PROGRAM CartControl
VAR
	// cart instance
	m_masterCart :FB_MasterCart;
	
	//cart related UI
	m_cartUIData : ST_CartUIData;
	
	// Output cart status
	m_cartStatus AT%Q* : ST_CartStatus;
	
	// Cart  joint data
	m_cartJointData AT %Q* :ST_CartJointData;
	
	// wait time before cart init for ethercat to be statble 
	m_cartInitWaitTime : LREAL:=0;
	
	// cart init flag
	m_cartInit :BOOL :=FALSE;
	
	m_workHeartTon0 : TON;
	m_workHeartTon1 : TON;
	
END_VAR

// wait communication to be stable
IF(m_cartInitWaitTime<g_robotInitWaitTime) THEN
	m_cartInitWaitTime := m_cartInitWaitTime+g_armCtrlCycleTime;
	RETURN;
END_IF

// cart init
IF m_cartInit =FALSE THEN
	m_masterCart.Init();
	m_cartInit:=TRUE;
END_IF

// input from UI
UIInputProcess();

// cart run
m_masterCart.run(m_cartUIData);

// status/joint data output
m_masterCart.getStatus(m_cartStatus, m_cartJointData);

// tranform data from UI(global variable write by ADS) to ST_UIData
METHOD UIInputProcess : BOOL
VAR_INPUT
END_VAR
//init cart joint postion
IF (GVL_interactUI.Upper_PC_Initial_Finished=FALSE) THEN
	GVL_interactUI.Upper_PC_Initial_Finished:=TRUE;
	//当前位置保存
	m_cartUIData.m_cmdCancelErgonPos := m_cartJointData.m_curJntPos;
	GVL_interactUI.g_ergonomicCtrlEnable.m_ergonInfoModify:=TRUE;//初始化时将台车现在的位置赋值给UI；
END_IF

IF  GVL_interactUI.g_ergonomicCtrlEnable.m_recovErgonEnable AND NOT GVL_interactUI.g_ergonomicCtrlEnableLast.m_recovErgonEnable THEN
	GVL_interactUI.g_ergonomicCtrlEnable.m_recovErgonFinshed:=FALSE;
	m_cartUIData.m_cmdCancelErgonPos := m_cartJointData.m_curJntPos;
	m_cartUIData.m_cmdJntPos[1] := GVL_interactUI.g_ergonomicCtrlData.m_monitorHeight;
	m_cartUIData.m_cmdJntPos[2] := GVL_interactUI.g_ergonomicCtrlData.m_headAngle;
	m_cartUIData.m_cmdJntPos[3] := GVL_interactUI.g_ergonomicCtrlData.m_handrailHeight;
	m_cartUIData.m_cmdJntPos[4] := GVL_interactUI.g_ergonomicCtrlData.m_footDistance;
	
END_IF
	m_cartUIData.m_ergonomicCrl.m_recovErgonEnable := GVL_interactUI.g_ergonomicCtrlEnable.m_recovErgonEnable;
	
IF (GVL_interactUI.g_ergonomicCtrlEnableLast.m_cancelRecovErgonEnable=FALSE) AND (GVL_interactUI.g_ergonomicCtrlEnable.m_cancelRecovErgonEnable=TRUE) THEN
	GVL_interactUI.g_ergonomicCtrlEnable.m_cancelRecovErgonFinshed:=FALSE;
	m_cartUIData.m_cmdJntPos := m_cartUIData.m_cmdCancelErgonPos;
END_IF
m_cartUIData.m_ergonomicCrl.m_cancelRecovErgonEnable := GVL_interactUI.g_ergonomicCtrlEnable.m_cancelRecovErgonEnable;

GVL_interactUI.g_ergonomicCtrlEnableLast:=GVL_interactUI.g_ergonomicCtrlEnable;
GVL_interactUI.g_ergonomicCtrlEnable.m_cancelRecovErgonFinshed := m_cartStatus.m_cancelErgonAdjustArrival;
GVL_interactUI.g_ergonomicCtrlEnable.m_recovErgonFinshed := m_cartStatus.m_ergonAdjustArrival;

GVL_interactUI.g_surgonHeadIn:=m_cartStatus.m_surgonReady;

GVL_interactUI.g_ergonomicCurData.m_monitorHeight := m_cartJointData.m_curJntPos[1];
GVL_interactUI.g_ergonomicCurData.m_headAngle := m_cartJointData.m_curJntPos[2];
GVL_interactUI.g_ergonomicCurData.m_handrailHeight := m_cartJointData.m_curJntPos[3];
GVL_interactUI.g_ergonomicCurData.m_footDistance:= m_cartJointData.m_curJntPos[4];



//work heart
m_workHeartTon0(IN:= GVL_interactUI.g_heartBeat = 1, PT:= T#1S, Q=> , ET=> );
m_workHeartTon1(IN:= GVL_interactUI.g_heartBeat = 0, PT:= T#1S, Q=> , ET=> );
IF m_workHeartTon0.Q THEN
	GVL_interactUI.g_heartBeat :=0 ;
ELSIF m_workHeartTon1.Q THEN
	GVL_interactUI.g_heartBeat  :=1 ;
END_IF
END_METHOD

END_PROGRAM

(* stored: Version 1.1.0.1, ProductVersion 3.1.4024.11
   POU CartControl: Id {c247957a-c15a-480d-acbc-bde71223345b}, SpecialFunc None
   Method UIInputProcess: Id {572b15b0-e408-437d-abc5-fa6c233e3112} *)
